FUNCTION_BLOCK E_SELECT (* Selection between two events *)
  (* Standard: 61499-1; Classification: Event processing *)
  (* Version 0.1, 2002-01-28, JHC, Rockwell Automation, XML version *)
  (* Version 0.0, 1997-12-05, JHC, Rockwell Automation, SRC version *)
  (* Compiler header: package fb.rt.events; *)
  (* Compiler Java IBM VisualAge 3.0 *)
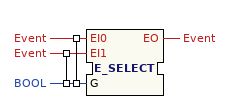
  EVENT_INPUT
    EI0 WITH G; (* Input event,selected when G=0 *)
    EI1 WITH G; (* Input event,selected when G=1 *)
  END_EVENT
  EVENT_OUTPUT
    EO; (* Output Event *)
  END_EVENT
  VAR_INPUT
    G : BOOL; (* Select EI0 when G=0,EI1 when G=1 *)
  END_VAR
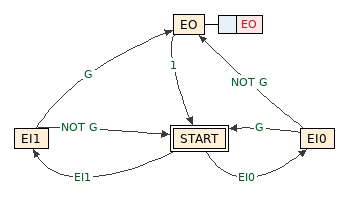
  EC_STATES
    START; (* Initial State *)
    EO : -> EO; (* Issue Output Event *)
    EI0; (* EI0 arrived *)
    EI1; (* EI1 arrived *)
  END_STATES
  EC_TRANSITIONS
    START TO EI0 := EI0;
    START TO EI1 := EI1;
    EI0 TO EO := NOT G;
    EI0 TO START := G;
    EI1 TO EO := G;
    EI1 TO START := NOT G;
    EO TO START := 1;
  END_TRANSITIONS
END_FUNCTION_BLOCK
